TYPE (* A service registry entry for the Arrowhead framework 4.0 *)
  (* Standard: 61499-2 *)
  (* Version 1.0, 2018-09-26, Jose Cabral, fortiss GmbH *)
  (* ASN.1 tag APPLICATION 1 *)
  ServiceRegistryEntry : STRUCT
    providedService : ArrowheadService; (* The Arrowhead Service object that is provided (SD and supported IDD-s) *)
    provider : ArrowheadSystem; (* ArrowheadSystem that is providing the Service *)
    serviceURI : WSTRING; (* The URL subpath of the Service within the address:port of the Provider *)
    version : DINT; (* The version numbering of the Service provided *)
    udp : BOOL; (* True, if the service is provided via UDP. By default, it is false *)
    ttl : DINT; (* Service validity time period expressed in seconds. This gets converted to a date-time, and stored in the database *)
    metadata : WSTRING; (* Metadata belonging to a service/provider pair *)
  END_STRUCT;
END_TYPE
